{attribute 'linkalways'} 
{attribute 'no_explicit_call' := 'This FB is a CLASS and must be accessed using methods or properties'}
{attribute 'enable_dynamic_creation'}
FUNCTION_BLOCK _Array0to3OfINT EXTENDS ArrayDatatypeBase_1D
VAR CONSTANT
	lBound : DINT := 0;
	uBound : DINT := 3;
END_VAR
VAR
	localData : ARRAY [lBound..uBound] OF INT;
	activeData : REFERENCE TO ARRAY [lBound..uBound] OF INT REF= localData;
	elements : ARRAY [lBound..uBound] OF _INT(0);
	baseType : _INT(0);
END_VAR

PROPERTY PUBLIC Address : PVOID
GET
Address := ADR(activeData);
END_GET
END_PROPERTY

PROPERTY PUBLIC BaseDatatype : I_Datatype
GET
BaseDatatype := baseType;
END_GET
END_PROPERTY

METHOD PUBLIC ClearReference
VAR_INPUT
END_VAR
activeData REF= localData;
SetElementReference();
END_METHOD

METHOD PUBLIC Clone : I_Datatype
VAR
    pClone : POINTER TO _Array0to3OfINT;
END_VAR
pClone := __NEW(_Array0to3OfINT());
pClone^.Value := Value;
Clone := pClone^;
END_METHOD

METHOD FB_init : BOOL
VAR_INPUT
	bInitRetains : BOOL; // if TRUE, the retain variables are initialized (warm start / cold start)
	bInCopyCode : BOOL;  // if TRUE, the instance afterwards gets moved into the copy code (online change)
END_VAR
SetElementReference();
END_METHOD

METHOD PUBLIC MakeReferenceTo
VAR_INPUT
	ReferenceTarget : REFERENCE TO ARRAY [lBound..uBound] OF INT;
END_VAR
activeData REF= ReferenceTarget;
SetElementReference();
END_METHOD

METHOD PROTECTED OnSerializeArrayValues
VAR_INPUT
	Serializer : I_Serializer;
END_VAR
VAR
	i : DINT;
END_VAR
FOR i := lBound TO uBound DO
	elements[i].SerializeWith(Serializer);
END_FOR
END_METHOD

METHOD PROTECTED SetElementReference
VAR_INPUT
END_VAR
VAR
	i : DINT;
END_VAR
FOR i := lBound TO uBound DO
	elements[i].MakeReferenceTo(activeData[i]);
END_FOR
END_METHOD

PROPERTY PUBLIC Size : UDINT
GET
Size := SIZEOF(activeData);
END_GET
END_PROPERTY

METHOD PROTECTED TryDeserializeArrayValues : BOOL
VAR_INPUT
	Deserializer : I_Deserializer;
	Feedback : I_DeserializerFeedback;
END_VAR
VAR
	enumerator : I_DeserializerArrayForwardEnumerator;
	i : DINT;
END_VAR
enumerator := Deserializer.GetArrayEnumerator();
i := lBound;

WHILE enumerator.MoveNext() AND i <= uBound DO
	
	IF NOT elements[i].TryDeserializeFrom(enumerator.Current, Feedback) THEN
		EXIT;
	END_IF
	i := i + 1;

END_WHILE
enumerator.Dispose();
END_METHOD

METHOD PUBLIC TryGetElementAsDatatypeByIndex : BOOL
VAR_INPUT
	Index : DINT;
	Destination : REFERENCE TO I_Datatype;
END_VAR
IF Index < lbound OR Index > ubound THEN
	RETURN;
END_IF

Destination := elements[Index];
TryGetElementAsDatatypeByIndex := TRUE;
END_METHOD

METHOD PUBLIC TryGetLowerBound : BOOL
VAR_INPUT
	Dimention : UDINT;
	Destination : REFERENCE TO DINT;
END_VAR
IF Dimention = 1 THEN
	Destination := lBound;
	TryGetLowerBound := TRUE;
END_IF
END_METHOD

METHOD PUBLIC TryGetUpperBound : BOOL
VAR_INPUT
	Dimention : UDINT;
	Destination : REFERENCE TO DINT;
END_VAR
IF Dimention = 1 THEN
	Destination := uBound;
	TryGetUpperBound := TRUE;
END_IF
END_METHOD

METHOD TryMakeReferenceTo : BOOL
VAR_INPUT
	Target : I_Datatype;
END_VAR
VAR
	pTargetData : POINTER TO ARRAY [lBound..uBound] OF INT;
END_VAR
IF NOT IsEquivalentTo(Target) THEN
	RETURN;
END_IF

pTargetData := Target.Address;
activeData REF= pTargetData^;
SetElementReference();
TryMakeReferenceTo := TRUE;
END_METHOD

PROPERTY PUBLIC Value : REFERENCE TO ARRAY [lBound..uBound] OF INT;
GET
Value ref= activeData;
END_GET
END_PROPERTY

END_FUNCTION_BLOCK

(* stored: Version 1.1.0.1, ProductVersion 3.1.4024.13
   POU _Array0to3OfINT: Id {6ccc462a-ba6f-06b7-2678-637ca8eee331}, SpecialFunc None
   Folder Core: Id {643bf541-16a0-0c27-3281-163285a1172a}
   Folder Constructor: Id {da4482b0-a3e7-0497-0bcd-afa0b2846ccf}
   Folder Protected: Id {dc462ef5-df94-0cf4-3c66-a752997ec461}
   Folder Customize: Id {630db994-5223-0c28-1cab-6708a25969c4}
   Property Address: Id {029a588f-930f-0d1b-072d-c86426f0d95a}
   Get Get: Id {c9d3cfbd-1914-0d03-0534-5f5f477efb4d}
   Property BaseDatatype: Id {ec9e06f2-1a0f-0494-0c73-8c20fb32aa84}
   Get Get: Id {693821ce-c408-017c-186f-77d7f9c4341d}
   Method ClearReference: Id {796badba-8ff0-0bee-2722-be9c6f0c419e}
   Method Clone: Id {f82e97a7-fccc-091d-1c96-29a4c28765cd}
   Method FB_init: Id {fe0c89a6-98d1-0e0b-2efe-ecae57c05507}
   Method MakeReferenceTo: Id {1a235b1e-9ed8-0987-38f4-d881c3f7c4df}
   Method OnSerializeArrayValues: Id {190351cd-1deb-07c8-0f56-d48a8c310415}
   Method SetElementReference: Id {32112e8a-024b-0071-0a7d-9bb2a1c3ff52}
   Property Size: Id {dee4d6ac-e635-08cc-18e6-d6161a02582a}
   Get Get: Id {c274940d-2d92-0146-3224-4a5975f1cd2b}
   Method TryDeserializeArrayValues: Id {23aa61bc-cb7a-0c2c-1488-6569a7723385}
   Method TryGetElementAsDatatypeByIndex: Id {c3e9b330-83e8-00e2-1611-03a80dbb54a7}
   Method TryGetLowerBound: Id {4d35bf74-4c6f-039e-295f-7eeab296365a}
   Method TryGetUpperBound: Id {81c627fc-9de7-0990-3d0b-f58a8e226607}
   Method TryMakeReferenceTo: Id {fcf5cc76-5628-0ccb-1441-5e29e31ced47}
   Property Value: Id {15770933-654c-035f-0e11-7fa51b87ee01}
   Get Get: Id {40a6dd7d-044f-0eae-1c98-58bb4b4d6727} *)
